FUNCTION_BLOCK FINAL FB_DolMotor EXTENDS FB_EventLogger 
VAR_INPUT
	Energized					: BOOL;								//Motor Energize Input
	InhibitFeedbackOn			: BOOL;								//Inhibit Feedback On Alarms
	InhibitFeedbackOff			: BOOL;								//Inhibit Feedback Off Alarms
	AutoEN						: BOOL;								//Auto mode enable
END_VAR                                                 			
VAR_IN_OUT                                              			
	Control						: ST_System;						//Machine Control Instance
END_VAR                                                 			
VAR                                                     			
	_AutoFwd					: BOOL;								//Auto of forward command
	_AutoRev					: BOOL;								//Auto of reverse command
	_ManSP1						: BOOL;								//Speed Selection 1
	_ManOnFwd					: BOOL;								//Manual on forwards
	_ManOnRev					: BOOL;								//Manual on reverse
	_ManOff						: BOOL;								//Manual Off
	_ForceOnFwd					: BOOL;								//Force on forward
	_ForceOnRev					: BOOL;								//Force on reverse
	_ForceOff					: BOOL;								//Force off
	_Fault						: BOOL;								//Fault
	_IsolatorFeedback    AT %I*	: BOOL;								//Motor Isolator feedback
	_RunFeedback		 AT %I*	: BOOL;								//Motor Running feedback input
	_OverloadFeedBack    AT %I* : BOOL;								//Motor Overload feedback Input
	_ValueFwd			 AT %Q*	: BOOL;								//Value (physical output)
	_ValueRev			 AT %Q*	: BOOL;								//Value (physical output)
	_ValueSP1			 AT %Q*	: BOOL;								//Value for Secondary Speed (physical output)
	_Velocity			 AT %Q*	: INT;								//Value for Analogue Speed Control (physical output)
	_Running					: BOOL;								//Motor is running
	_MotorOn_ET					: REAL;								//Time output has been on since last being off (sec)
	_FaultTimer_ET				: REAL;								//Fault timer elapsed (sec)
	_Alarm						: BOOL;								//Device Alarm
	_Warning					: BOOL;								//Device Warning
	_AlarmNum					: DINT;								//Device Alarm Number
	_WarningNum					: DINT;								//Device Warning Number
	_R_Trig						: ARRAY[0..9] OF R_TRIG;			//Private Rising Edge Triggers
END_VAR
VAR PERSISTENT
	_Name						: STRING[15];						//Name for HMI
	_Description				: STRING[40];						//Description for HMI
	_AlarmMute					: BOOL;								//Alarm Mute
	_TotalMotorOnHours			: REAL;								//Total Amount of run hours
	_TypeConfig					: SINT;								//0 = DOL Normal, 1 = DOL Reversing
	_StartTimer_PT				: REAL;								//Start Timer Preset
	_FaultTimer_PT				: REAL;								//Fault timer preset time
	_Variables					: ARRAY [0..9] OF ST_Variable;		//Device Associated Varibles Array		
END_VAR

M_AlarmMonitor();
M_WarningMonitor();
M_UnlatchManuals();
M_MotorOutputs();

//Run hours
IF Control.Inputs.HoursReset THEN
	_TotalMotorOnHours := 0;
END_IF
IF _ValueFwd OR _ValueRev THEN
	_MotorOn_ET :=_MotorOn_ET + Control.SystemTime.ScanTime;
ELSE
	_TotalMotorOnHours :=_TotalMotorOnHours + (_MotorOn_ET / 3600);
	_MotorOn_ET := 0;
END_IF

//Motor startup timer
IF (_MotorOn_ET >_StartTimer_PT) THEN
	_Running := TRUE;
ELSE
	_Running := FALSE;
END_IF

{attribute 'monitoring' := 'variable'}
PROPERTY PUBLIC Alarm : Bool
GET
Alarm := _Alarm;
END_GET
END_PROPERTY

{attribute 'monitoring' := 'variable'}
PROPERTY PUBLIC AlarmMute : BOOL
SET
_AlarmMute := AlarmMute;
END_SET
END_PROPERTY

{attribute 'monitoring' := 'variable'}
PROPERTY PUBLIC AutoFwd : BOOL
GET // PUBLIC
AutoFwd := _AutoFwd;
END_GET
SET
_AutoFwd := AutoFwd;
END_SET
END_PROPERTY

{attribute 'monitoring' := 'variable'}
PROPERTY PUBLIC AutoRev : BOOL
GET // PUBLIC
AutoRev := _AutoRev;
END_GET
SET
_AutoRev := AutoRev;
END_SET
END_PROPERTY

{attribute 'monitoring' := 'variable'}
PROPERTY PUBLIC Description : String[40]
GET
Description := _Description;
END_GET
SET
_Description := Description;
END_SET
END_PROPERTY

{attribute 'monitoring' := 'variable'}
PROPERTY PUBLIC Fault : Bool
SET
_Fault := Fault;
END_SET
END_PROPERTY

{attribute 'monitoring' := 'variable'}
PROPERTY PUBLIC FaultTimer_PT : real
GET
FaultTimer_PT := _FaultTimer_PT;
END_GET
SET
_FaultTimer_PT := FaultTimer_PT;
END_SET
END_PROPERTY

{attribute 'monitoring' := 'variable'}
PROPERTY PUBLIC ForceOff : Bool
GET
ForceOff := _ForceOff;
END_GET
SET
_ForceOff := ForceOff;
END_SET
END_PROPERTY

{attribute 'monitoring' := 'variable'}
PROPERTY PUBLIC ForceOnFwd : Bool
GET
ForceOnFwd := _ForceOnFwd;
END_GET
SET
_ForceOnFwd := ForceOnFwd;
END_SET
END_PROPERTY

{attribute 'monitoring' := 'variable'}
PROPERTY PUBLIC ForceOnRev : Bool
GET
ForceOnRev := _ForceOnRev;
END_GET
SET
_ForceOnRev := ForceOnRev;
END_SET
END_PROPERTY

{attribute 'monitoring' := 'variable'}
PROPERTY PUBLIC IsolatorFeedback : BOOL
GET // PUBLIC
IsolatorFeedback := _IsolatorFeedback;
END_GET
SET
_IsolatorFeedback := IsolatorFeedback;
END_SET
END_PROPERTY

METHOD PRIVATE M_AlarmMonitor
VAR_INPUT
END_VAR
VAR_INST
END_VAR
VAR_INST // added by the converter: edge detectors and wires of the graphical bodies
    _w1, _w2, _w3, _w4, _w5 : BOOL;
END_VAR
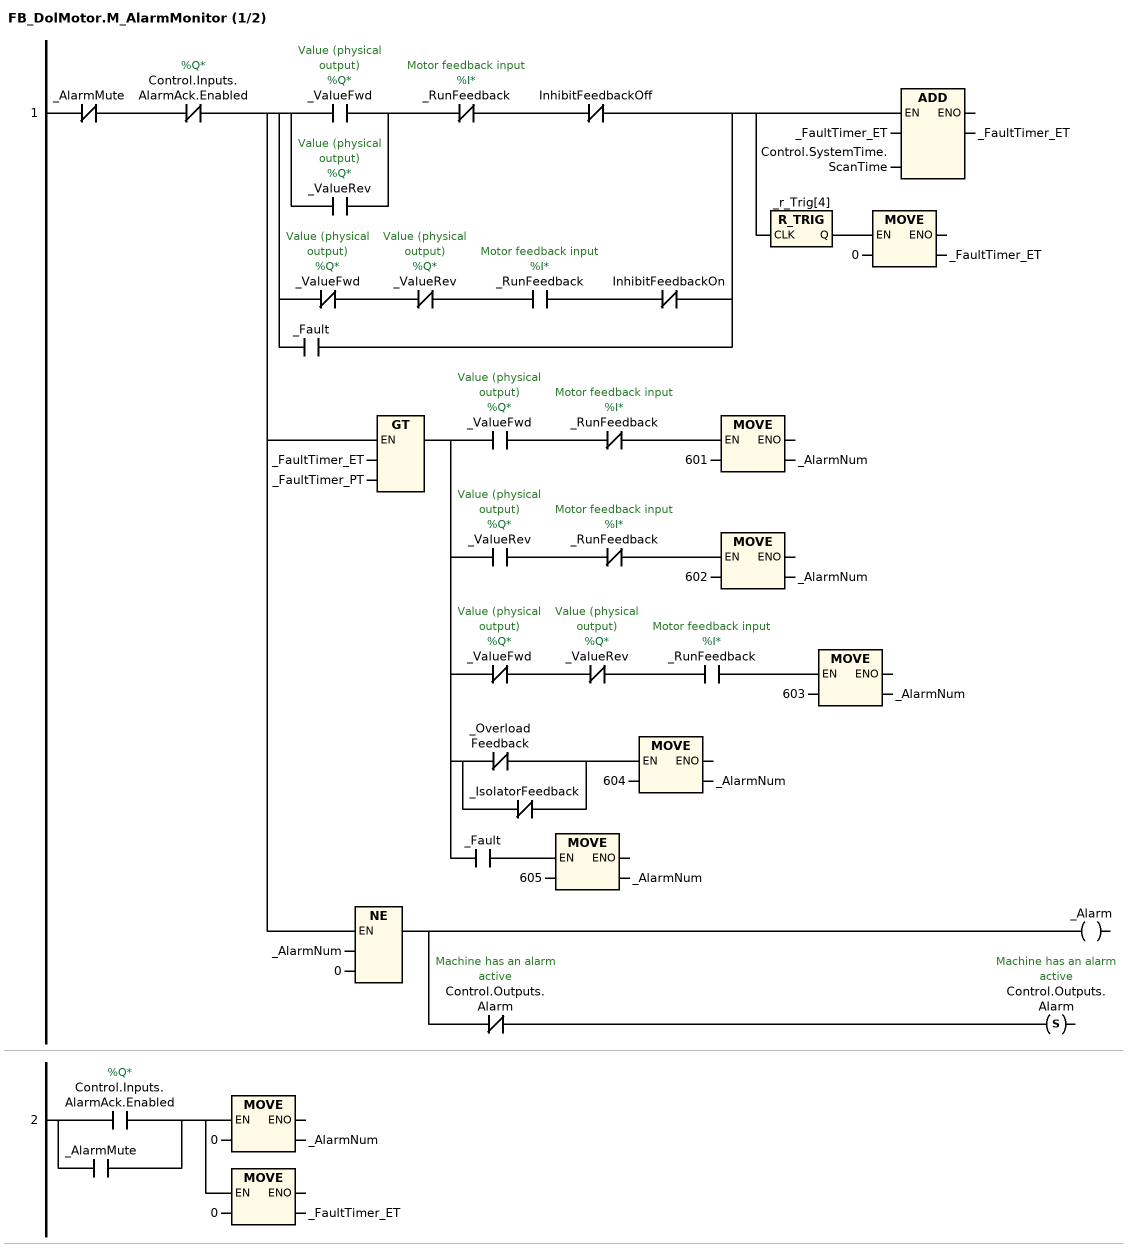
// NETWORK 1
//   Control.Inputs.AlarmAck.Enabled: AT %Q*
//   _ValueFwd: Value (physical output) | AT %Q*
//   _ValueRev: Value (physical output) | AT %Q*
//   _RunFeedback: Motor feedback input | AT %I*
//   _FaultTimer_ET: Fault timer elapsed (sec)
//   Control.SystemTime.ScanTime: Last scan time (Seconds)
//   Control.Outputs.Alarm: Machine has an alarm active
_w1 := NOT _AlarmMute AND NOT Control.Inputs.AlarmAck.Enabled;
_w2 := _w1 AND ((_ValueFwd OR _ValueRev) AND NOT _RunFeedback AND NOT InhibitFeedbackOff OR NOT _ValueFwd AND NOT _ValueRev AND _RunFeedback AND NOT InhibitFeedbackOn OR _Fault);
IF _w2 THEN _FaultTimer_ET := _FaultTimer_ET + Control.SystemTime.ScanTime; END_IF
_r_Trig[4](CLK := _w2); // R_TRIG
IF _r_Trig[4].Q THEN _FaultTimer_ET := 0; END_IF
_w3 := _w1 AND _FaultTimer_ET > _FaultTimer_PT;
IF _w3 AND _ValueFwd AND NOT _RunFeedback THEN _AlarmNum := 601; END_IF
IF _w3 AND _ValueRev AND NOT _RunFeedback THEN _AlarmNum := 602; END_IF
IF _w3 AND NOT _ValueFwd AND NOT _ValueRev AND _RunFeedback THEN _AlarmNum := 603; END_IF
IF _w3 AND (NOT _OverloadFeedback OR NOT _IsolatorFeedback) THEN _AlarmNum := 604; END_IF
IF _w3 AND _Fault THEN _AlarmNum := 605; END_IF
_w4 := _w1 AND _AlarmNum <> 0;
_Alarm := _w4;
Control.Outputs.Alarm S= _w4 AND NOT Control.Outputs.Alarm;

// NETWORK 2
//   Control.Inputs.AlarmAck.Enabled: AT %Q*
//   _FaultTimer_ET: Fault timer elapsed (sec)
_w5 := Control.Inputs.AlarmAck.Enabled OR _AlarmMute;
IF _w5 THEN _AlarmNum := 0; END_IF
IF _w5 THEN _FaultTimer_ET := 0; END_IF

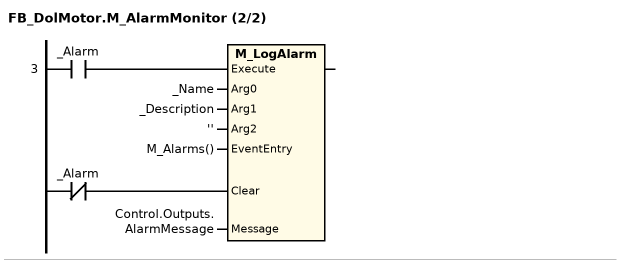
// NETWORK 3
M_LogAlarm(Execute := _Alarm, Arg0 := _Name, Arg1 := _Description, Arg2 := '', EventEntry := M_Alarms(), Clear := NOT _Alarm, Message := Control.Outputs.AlarmMessage);
END_METHOD

METHOD PRIVATE M_Alarms : TcEventEntry
VAR_INPUT
END_VAR
VAR_INST
END_VAR
CASE _AlarmNum OF
601:    M_Alarms :=   TC_Events.TcDolMotor.A_601;//Forward Feedback OFF Alarm
602:    M_Alarms :=   TC_Events.TcDolMotor.A_602;//Reverse Feedback OFF Alarm
603:    M_Alarms :=   TC_Events.TcDolMotor.A_603;//Feedback ON Alarm
604:    M_Alarms :=   TC_Events.TcDolMotor.A_604;//External Feedback Alarm
605:    M_Alarms :=   TC_Events.TcDolMotor.A_605;//Drive Fault
ELSE           
		M_Alarms :=   TC_Events.TcDolMotor.A_Undefined;
END_CASE
END_METHOD

METHOD PRIVATE M_MotorOutputs
VAR_INPUT
END_VAR
VAR_INST
	_Fwd	: BOOL;
	_Rev	: BOOL;
END_VAR
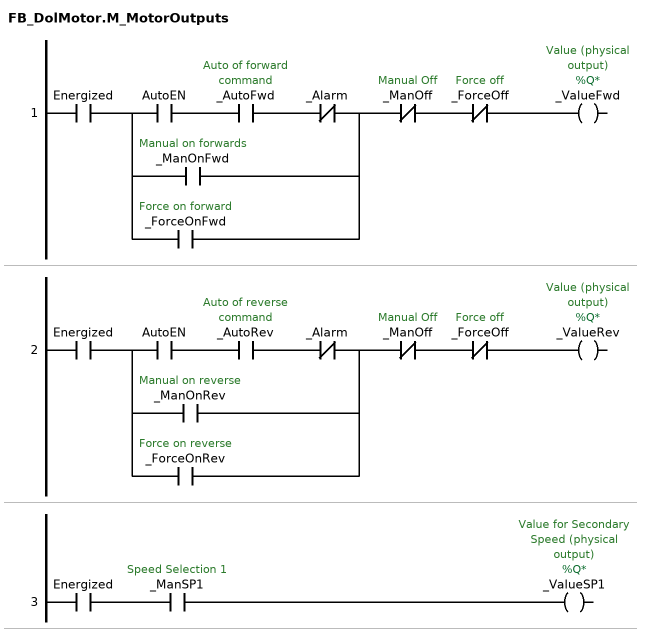
// NETWORK 1
//   _AutoFwd: Auto of forward command
//   _ManOnFwd: Manual on forwards
//   _ForceOnFwd: Force on forward
//   _ManOff: Manual Off
//   _ForceOff: Force off
//   _ValueFwd: Value (physical output) | AT %Q*
_ValueFwd := Energized AND (AutoEN AND _AutoFwd AND NOT _Alarm OR _ManOnFwd OR _ForceOnFwd) AND NOT _ManOff AND NOT _ForceOff;

// NETWORK 2
//   _AutoRev: Auto of reverse command
//   _ManOnRev: Manual on reverse
//   _ForceOnRev: Force on reverse
//   _ManOff: Manual Off
//   _ForceOff: Force off
//   _ValueRev: Value (physical output) | AT %Q*
_ValueRev := Energized AND (AutoEN AND _AutoRev AND NOT _Alarm OR _ManOnRev OR _ForceOnRev) AND NOT _ManOff AND NOT _ForceOff;

// NETWORK 3
//   _ManSP1: Speed Selection 1
//   _ValueSP1: Value for Secondary Speed (physical output) | AT %Q*
_ValueSP1 := Energized AND _ManSP1;
END_METHOD

METHOD PRIVATE M_UnlatchManuals
VAR_INPUT
END_VAR
VAR_INST
END_VAR
VAR_INST // added by the converter: edge detectors and wires of the graphical bodies
    _rt1, _rt2, _rt3, _rt4 : R_TRIG;
END_VAR
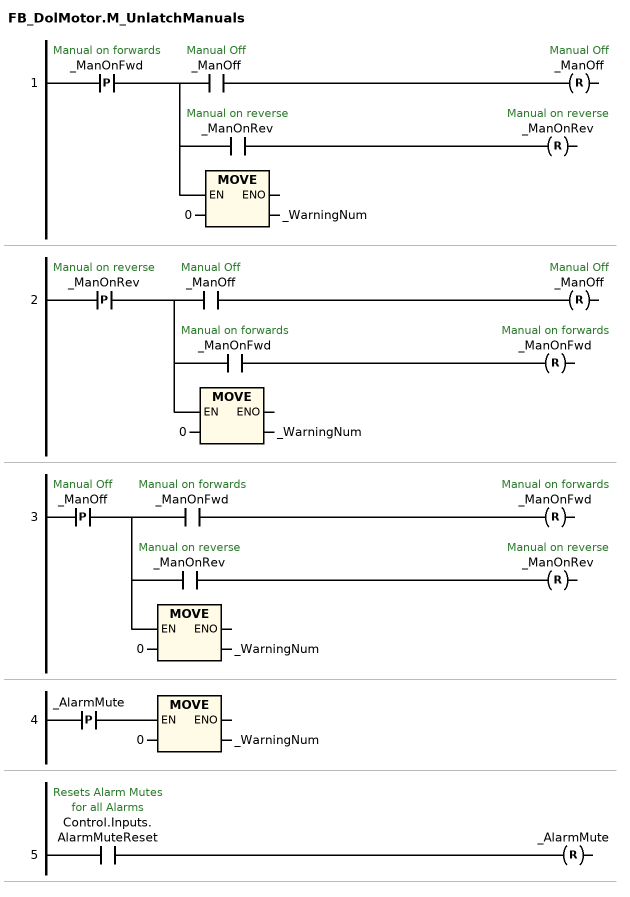
// NETWORK 1
//   _ManOnFwd: Manual on forwards
//   _ManOff: Manual Off
//   _ManOnRev: Manual on reverse
_rt1(CLK := _ManOnFwd);
_ManOff R= _rt1.Q AND _ManOff;
_ManOnRev R= _rt1.Q AND _ManOnRev;
IF _rt1.Q THEN _WarningNum := 0; END_IF

// NETWORK 2
//   _ManOnRev: Manual on reverse
//   _ManOff: Manual Off
//   _ManOnFwd: Manual on forwards
_rt2(CLK := _ManOnRev);
_ManOff R= _rt2.Q AND _ManOff;
_ManOnFwd R= _rt2.Q AND _ManOnFwd;
IF _rt2.Q THEN _WarningNum := 0; END_IF

// NETWORK 3
//   _ManOff: Manual Off
//   _ManOnFwd: Manual on forwards
//   _ManOnRev: Manual on reverse
_rt3(CLK := _ManOff);
_ManOnFwd R= _rt3.Q AND _ManOnFwd;
_ManOnRev R= _rt3.Q AND _ManOnRev;
IF _rt3.Q THEN _WarningNum := 0; END_IF

// NETWORK 4
_rt4(CLK := _AlarmMute);
IF _rt4.Q THEN _WarningNum := 0; END_IF

// NETWORK 5
//   Control.Inputs.AlarmMuteReset: Resets Alarm Mutes for all Alarms
_AlarmMute R= Control.Inputs.AlarmMuteReset;
END_METHOD

METHOD PRIVATE M_WarningMonitor
VAR_INPUT
END_VAR
VAR_INST
END_VAR
VAR_INST // added by the converter: edge detectors and wires of the graphical bodies
    _w1, _w2 : BOOL;
END_VAR
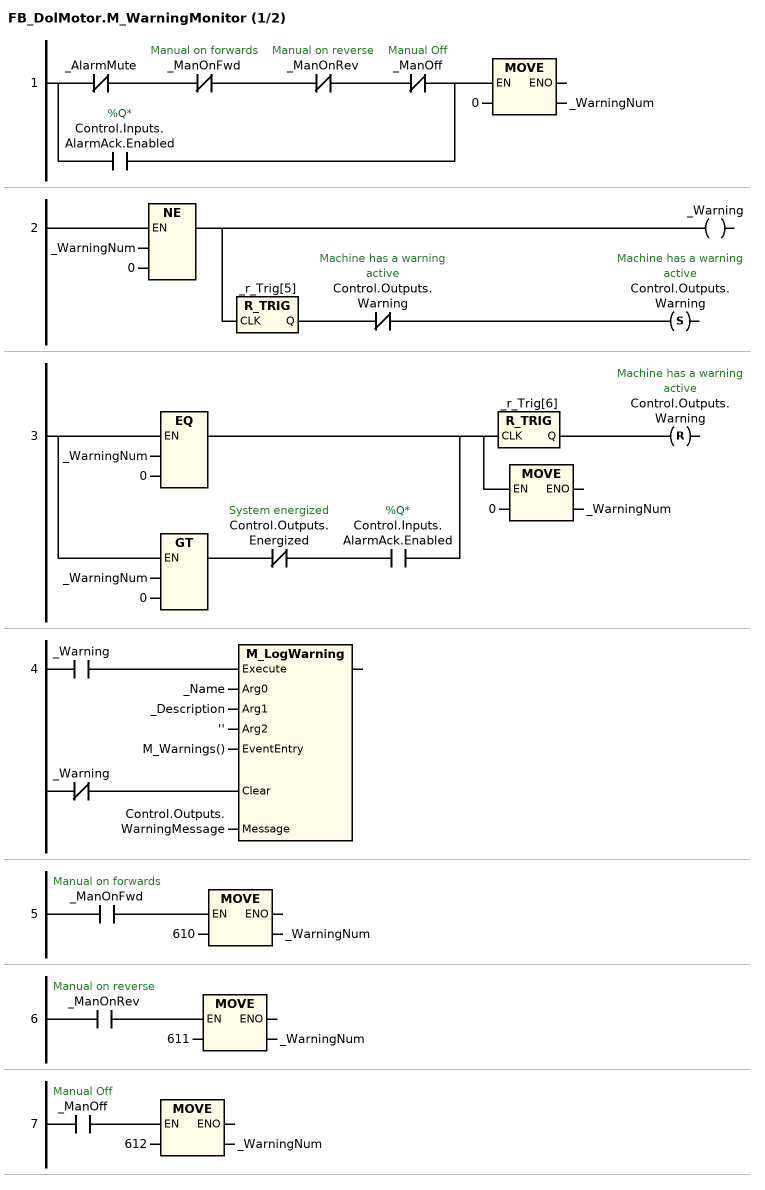
// NETWORK 1
//   _ManOnFwd: Manual on forwards
//   _ManOnRev: Manual on reverse
//   _ManOff: Manual Off
//   Control.Inputs.AlarmAck.Enabled: AT %Q*
IF NOT _AlarmMute AND NOT _ManOnFwd AND NOT _ManOnRev AND NOT _ManOff OR Control.Inputs.AlarmAck.Enabled THEN
    _WarningNum := 0;
END_IF

// NETWORK 2
//   Control.Outputs.Warning: Machine has a warning active
_w1 := _WarningNum <> 0;
_Warning := _w1;
_r_Trig[5](CLK := _w1); // R_TRIG
Control.Outputs.Warning S= _r_Trig[5].Q AND NOT Control.Outputs.Warning;

// NETWORK 3
//   Control.Outputs.Energized: System energized
//   Control.Inputs.AlarmAck.Enabled: AT %Q*
//   Control.Outputs.Warning: Machine has a warning active
_w2 := _WarningNum = 0 OR _WarningNum > 0 AND NOT Control.Outputs.Energized AND Control.Inputs.AlarmAck.Enabled;
_r_Trig[6](CLK := _w2); // R_TRIG
Control.Outputs.Warning R= _r_Trig[6].Q;
IF _w2 THEN _WarningNum := 0; END_IF

// NETWORK 4
M_LogWarning(Execute := _Warning, Arg0 := _Name, Arg1 := _Description, Arg2 := '', EventEntry := M_Warnings(), Clear := NOT _Warning, Message := Control.Outputs.WarningMessage);

// NETWORK 5
//   _ManOnFwd: Manual on forwards
IF _ManOnFwd THEN _WarningNum := 610; END_IF

// NETWORK 6
//   _ManOnRev: Manual on reverse
IF _ManOnRev THEN _WarningNum := 611; END_IF

// NETWORK 7
//   _ManOff: Manual Off
IF _ManOff THEN _WarningNum := 612; END_IF

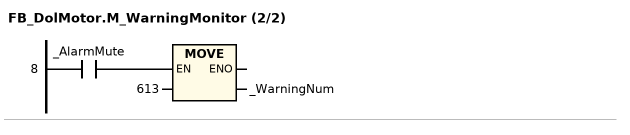
// NETWORK 8
IF _AlarmMute THEN _WarningNum := 613; END_IF
END_METHOD

METHOD PRIVATE M_Warnings : TcEventEntry
VAR_INPUT
END_VAR
VAR_INST
END_VAR
CASE _WarningNum OF
610:    M_Warnings :=   	TC_Events.TcDolMotor.W_610;//Manual ON Enabled
611:    M_Warnings :=   	TC_Events.TcDolMotor.W_611;//Manual Reverse Enabled				
612:    M_Warnings :=   	TC_Events.TcDolMotor.W_612;//Manual OFF Enabled		
613:    M_Warnings :=   	TC_Events.TcDolMotor.W_613;//Alarm Mute Active
ELSE             
		M_Warnings := 	   TC_Events.TcDolMotor.W_Undefined;	
END_CASE
END_METHOD

{attribute 'monitoring' := 'variable'}
PROPERTY PUBLIC ManOff : Bool
GET
ManOff := _ManOff;
END_GET
SET
_ManOff := ManOff;
END_SET
END_PROPERTY

{attribute 'monitoring' := 'variable'}
PROPERTY PUBLIC ManOnFwd : Bool
GET
ManOnFwd := _ManOnFwd;
END_GET
SET
_ManOnFwd := ManOnFwd;
END_SET
END_PROPERTY

{attribute 'monitoring' := 'variable'}
PROPERTY PUBLIC ManOnRev : Bool
GET
ManOnRev := _ManOnRev;
END_GET
SET
_ManOnRev := ManOnRev;
END_SET
END_PROPERTY

{attribute 'monitoring' := 'variable'}
PROPERTY PUBLIC ManSP1 : BOOL
GET // PUBLIC
_ManSP1 := ManSP1;
END_GET
SET
_ManSP1 := ManSP1;
END_SET
END_PROPERTY

{attribute 'monitoring' := 'variable'}
PROPERTY PUBLIC MotorOn_ET : real
GET
MotorOn_ET := _MotorOn_ET;
END_GET
END_PROPERTY

{attribute 'monitoring' := 'variable'}
PROPERTY PUBLIC Name : String[15]
GET
Name := _Name;
END_GET
SET
_Name := Name;
END_SET
END_PROPERTY

{attribute 'monitoring' := 'variable'}
PROPERTY PUBLIC OverloadFeedback : BOOL
GET // PUBLIC
OverloadFeedback := _OverloadFeedback;
END_GET
SET
_OverloadFeedback := OverloadFeedback;
END_SET
END_PROPERTY

{attribute 'monitoring' := 'variable'}
PROPERTY PUBLIC RunFeedback : BOOL
GET // PUBLIC
RunFeedback := _RunFeedback;
END_GET
SET
_RunFeedback := RunFeedback;
END_SET
END_PROPERTY

{attribute 'monitoring' := 'variable'}
PROPERTY PUBLIC Running : Bool
GET
Running := _Running;
END_GET
END_PROPERTY

{attribute 'monitoring' := 'variable'}
PROPERTY PUBLIC StandbyReset : Bool
GET
StandbyReset := _ForceOff;
END_GET
SET
_ForceOff := StandbyReset;
END_SET
END_PROPERTY

{attribute 'monitoring' := 'variable'}
PROPERTY PUBLIC StartTimer_PT : real
GET
StartTimer_PT := _StartTimer_PT;
END_GET
SET
_StartTimer_PT := StartTimer_PT;
END_SET
END_PROPERTY

{attribute 'monitoring' := 'variable'}
PROPERTY PUBLIC TotalMotorOnHours : real
GET
TotalMotorOnHours := _TotalMotorOnHours;
END_GET
END_PROPERTY

{attribute 'monitoring' := 'variable'}
PROPERTY PUBLIC TypeConfig : sint
SET
_TypeConfig := TypeConfig;
END_SET
END_PROPERTY

{attribute 'monitoring' := 'variable'}
PROPERTY PUBLIC ValueFwd : BOOL
GET // PUBLIC
ValueFwd := _ValueFwd;
END_GET
SET
_ValueFwd := ValueFwd;
END_SET
END_PROPERTY

{attribute 'monitoring' := 'variable'}
PROPERTY PUBLIC ValueRev : BOOL
GET // PUBLIC
ValueRev := _ValueRev;
END_GET
SET
_ValueRev := ValueRev;
END_SET
END_PROPERTY

PROPERTY PUBLIC Variables : REFERENCE TO ARRAY[0..9] OF ST_Variable
GET
Variables REF= _Variables;
END_GET
END_PROPERTY

{attribute 'monitoring' := 'variable'}
PROPERTY PUBLIC Velocity : INT
GET
Velocity:= _Velocity;
END_GET
SET
_Velocity:= Velocity;
END_SET
END_PROPERTY

{attribute 'monitoring' := 'variable'}
PROPERTY PUBLIC Warning : Bool
GET
Warning := _Warning;
END_GET
END_PROPERTY

END_FUNCTION_BLOCK

(* stored: Version 1.1.0.1, ProductVersion 3.1.4024.3
   POU FB_DolMotor: Id {78f45cf4-15cb-4352-8aa4-cf663d7bc5af}, SpecialFunc None
   Property Alarm: Id {9547deec-586e-4ceb-9356-ce97db5cd6ce}
   Get Get: Id {ffb2bcc9-b83a-45ef-9a3d-a50aed37c0ae}
   Property AlarmMute: Id {4a0c68bd-30b9-4749-a5fd-bafc809ed34b}
   Set Set: Id {e2be9d0a-9212-456e-9f65-188ce6ae15e6}
   Property AutoFwd: Id {b62ead48-a769-4020-8a65-b60b11c60d4f}
   Get Get: Id {7602c8fc-124a-4a7f-a84e-f563cbe00199}
   Set Set: Id {13d1eb2a-c488-4100-9362-faef0ac720c7}
   Property AutoRev: Id {aad54209-b6c7-4315-ad29-9a2908ed2c8c}
   Get Get: Id {caea413d-7aef-4059-8920-09a840584040}
   Set Set: Id {52956703-a00b-40a6-a6cb-cde27136ac7b}
   Property Description: Id {c230680d-2437-4de2-9a5c-7a728a6c6b0c}
   Get Get: Id {9adfb88c-8ade-4272-8f6f-1e482da27e02}
   Set Set: Id {b05a44b2-dbeb-42de-ba1e-eebe438f2a58}
   Property Fault: Id {95a30caf-3e18-461e-86ef-93885530ca61}
   Set Set: Id {debbf8d8-fa81-43fa-ae15-7dc1c79fb739}
   Property FaultTimer_PT: Id {d8d3380d-2fd9-46e6-99ee-55de77a964fa}
   Get Get: Id {03c75602-60c6-49e3-a563-54fe532ace29}
   Set Set: Id {d810e762-5433-40c6-9be4-75dbbb876654}
   Property ForceOff: Id {7de45c4c-db81-45ca-8557-5ddf9919a567}
   Get Get: Id {bed74665-4d85-44f3-94ea-c09533ef250d}
   Set Set: Id {ccaf537e-89df-4623-a03f-5d352051f747}
   Property ForceOnFwd: Id {2bb7fa26-e52c-4326-bde3-dca99f5f8efa}
   Get Get: Id {43230645-4bbb-4092-a3ed-932f029a6eb6}
   Set Set: Id {f9632afd-7a93-42c5-870b-c92b60708739}
   Property ForceOnRev: Id {06b25ee0-c37d-483e-9e74-025190f6ce1c}
   Get Get: Id {1877a51b-496f-417e-98cc-db9d3bb880aa}
   Set Set: Id {40e66d6e-4fa6-4f7f-b6da-e432f2924c13}
   Property IsolatorFeedback: Id {4f9658c4-d639-4740-8250-aeb4b252c838}
   Get Get: Id {ca60ff3c-7e99-4dd5-b5e5-fdc6025f4ece}
   Set Set: Id {879280ff-b89a-4a87-9684-c839544e88ec}
   Method M_AlarmMonitor: Id {0dc40ea3-a0c4-425d-989f-bf1e868e0329}
   Method M_Alarms: Id {47413ca8-950f-4f1d-8bb7-640166c4ff83}
   Method M_MotorOutputs: Id {4522a35f-315f-41f1-a3e7-b1603eb6e316}
   Method M_UnlatchManuals: Id {77f81cd9-40dd-4a78-b42a-3f0dd21dd1fb}
   Method M_WarningMonitor: Id {b0db2067-3eeb-43db-8fb6-d1e75318db46}
   Method M_Warnings: Id {6500730e-6ea5-4dc7-9c58-4742da3295cf}
   Property ManOff: Id {afd9c3df-0ffc-45f7-b256-b5115605a0d7}
   Get Get: Id {470ebe66-c7a2-4e01-b602-652b7c133185}
   Set Set: Id {c182d924-312d-44b4-aa94-46eec861840a}
   Property ManOnFwd: Id {41f33f51-a9f6-4ae8-a238-7b2c27ed1da7}
   Get Get: Id {98625fda-08ce-4eee-8f31-31fea710aee0}
   Set Set: Id {dc0e4858-665e-46ac-ae93-640704fe2c99}
   Property ManOnRev: Id {99a510cb-8f0d-4e84-b526-29674a304325}
   Get Get: Id {95ad9dba-b49a-4b7e-b342-d6b1cf1aefae}
   Set Set: Id {eb70b4f5-bafb-49e7-b464-8e48cf3ad496}
   Property ManSP1: Id {a3674ddf-76e3-4b81-a5e3-0223b4b3bc70}
   Get Get: Id {3fd2f6e5-5ab3-4915-8e7a-0d0572797156}
   Set Set: Id {5e7208ab-47e5-4e35-9388-5d6ec8d56be4}
   Property MotorOn_ET: Id {8d1faebe-9b7c-430c-a488-b6ec59c5c2fd}
   Get Get: Id {85880e66-13e0-4247-b863-e9f4137f8e5d}
   Property Name: Id {d3638199-4b9c-44ed-b5dd-c7e554b034c6}
   Get Get: Id {b027419f-1bb5-4221-bf3e-972d7c329f20}
   Set Set: Id {331d7218-a578-4763-a5e5-a3a7d5739dc0}
   Property OverloadFeedback: Id {f3d26427-dd9f-4fea-826d-2db76b0115ab}
   Get Get: Id {65ae5917-ad2e-460b-9b99-11d2b7be7cee}
   Set Set: Id {4965bb7d-c838-402d-9c61-175b5975851f}
   Property RunFeedback: Id {7e5d2535-408b-4bc5-b108-d05fdc933b43}
   Get Get: Id {eed4a3d4-79ac-4645-9193-d6bd8fc133d6}
   Set Set: Id {228bc140-c33f-40c4-bdce-edeed79b6b09}
   Property Running: Id {d85736f8-0b4c-47d5-89cb-848876cc0660}
   Get Get: Id {fb1c62e6-d0c7-4433-9bda-bd1d16db4f30}
   Property StandbyReset: Id {7856710f-e696-4625-bef6-d4a1617ece2f}
   Get Get: Id {c09fb2ac-9857-4ad8-8f93-37a7d8dd8daf}
   Set Set: Id {43144911-f332-4380-825b-cb73fdfb5c1e}
   Property StartTimer_PT: Id {a5baa175-44e9-4fdb-ab79-6e6207642a9b}
   Get Get: Id {b5128e91-11b6-439a-a284-578bacf2073e}
   Set Set: Id {574ad21d-a161-4adc-aae7-b8eaf9c40651}
   Property TotalMotorOnHours: Id {336a1884-bc71-498e-9483-b3a5fa7b1d8a}
   Get Get: Id {5c2ca8ec-7093-4ecf-86be-07b76b5d296b}
   Property TypeConfig: Id {693ebf59-9fd1-4066-b4df-4e03e94f87ae}
   Set Set: Id {1a96f031-b871-4b1e-bbe2-42f7460bec31}
   Property ValueFwd: Id {2fb490af-853d-4286-949e-3beb13bc2921}
   Get Get: Id {aff7867a-2f81-49a9-ab58-2e55834fd0ec}
   Set Set: Id {b4780ab4-d9e2-4b8a-bd01-ce8a7508755d}
   Property ValueRev: Id {d8b54dcc-30ea-4c84-aa34-6ebac6b1f9af}
   Get Get: Id {9d7a65c1-3e5c-475e-b13b-03902b849dde}
   Set Set: Id {fc289996-aedb-4d35-97f1-e3f8f70b1944}
   Property Variables: Id {2576607e-144d-4da9-aaa4-b1e25509275d}
   Get Get: Id {3ca24952-129d-44b8-acbb-53b4fd870406}
   Property Velocity: Id {7ef902fd-f209-42e1-a853-b3df85f1813a}
   Get Get: Id {fb794f38-3b5c-43df-82a0-45958e123c90}
   Set Set: Id {919f2f32-8895-4eb4-8799-866a4f927f88}
   Property Warning: Id {5d28bd34-1400-483d-8344-71f477a2b184}
   Get Get: Id {4faa16c0-2769-4f54-b9e5-dd18dafedaee} *)
